Universal Robots URScript: extcontrol.script

def unnamed():
  set_tcp(p[0.0,0.0,0.0,0.0,0.0,0.0])
  set_payload(0.0)
  set_gravity([0.0, 0.0, 9.82])
  set_standard_analog_input_domain(0, 1)
  set_standard_analog_input_domain(1, 1)
  set_tool_analog_input_domain(0, 1)
  set_tool_analog_input_domain(1, 1)
  set_analog_outputdomain(0, 0)
  set_analog_outputdomain(1, 0)
  set_tool_voltage(0)
  set_input_actions_to_default()
  set_safety_mode_transition_hardness(1)
  set_tool_communication(False, 115200, 0, 1, 1.5, 3.5)
  set_tool_output_mode(0)
  set_tool_digital_output_mode(0, 1)
  set_tool_digital_output_mode(1, 1)
  # begin: URCap Installation Node
  #   Source: External Control, 1.0.4, FZI Research Center for Information Technology
  #   Type: External Control
  # end: URCap Installation Node
  while (True):
    $ 1 "Robot Program"
    # begin: URCap Program Node
    #   Source: External Control, 1.0.4, FZI Research Center for Information Technology
    #   Type: External Control
    $ 2 "Control by 192.168.56.1"
popup("The connection to the remote PC at 192.168.56.1:50002 could not be established. Reason: connect timed out","Receive program failed", False, True, blocking=True)
sync()    # end: URCap Program Node
  end
end
